// SIMATIC STEP 7 (V5.x) project Паллетайзер №2
// CPU: CPU 312
// station: P_ADR_BUS
// station: Hardware
// station: SIMATIC 300 Station
// program: S7 Program(2)

SYMBOL_TABLE
"FC2"	FC 2	FC 2	// Ручное управление
"FC3"	FC 3	FC 3	// Автоматическое управление
"КН1"	I 0.0	BOOL	// Кнопка ПУСК ВПЕРЕД устройства поддержания прокладки
"КН2"	I 0.1	BOOL	// Кнопка ПУСК НАЗАД устройства поддержания прокладки
"КН3"	I 0.2	BOOL	// Кнопка ПУСК ВПЕРЕД передвижная рама
"КН4"	I 0.3	BOOL	// Кнопка ПУСК НАЗАД передвижная рама
"КН5"	I 0.4	BOOL	// Кнопка ПУСК ВВЕРХ блокировка банок
"КН6"	I 0.5	BOOL	// Кнопка ПУСК ВНИЗ блокировка банок
"КН7"	I 0.6	BOOL	// Кнопка ПУСК ВВЕРХ штабелирующий лифт
"КН8"	I 0.7	BOOL	// Кнопка ПУСК ВНИЗ штабелирующий лифт
"КН9"	I 1.0	BOOL	// Кнопка ПУСК ВПЕРЕД выталкиватель
"КН10"	I 1.1	BOOL	// Кнопка ПУСК НАЗАД выталкиватель
"КН11"	I 1.2	BOOL	// Кнопка ПУСК ВВЕРХ лифт для паллет
"КН12"	I 1.3	BOOL	// Кнопка ПУСК ВНИЗ лифт для паллет
"6КВ1"	I 1.4	BOOL	// Лифт для паллет ВЕРХНЕЕ положение
"6КВ2"	I 1.5	BOOL	// Лифт для паллет НИЖНЕЕ положение
"КН15"	I 1.6	BOOL	// Кнопка ПУСК конвейера
"КН16"	I 1.7	BOOL	// Кнопка СТОП конвейера
"ПН17"	I 4.0	BOOL	// Переключатель РУЧНОЕ-АВТОМАТ
"КН18"	I 4.1	BOOL	// Кнопка ПУСК в автоматическом режиме
"КН17"	I 4.2	BOOL	// Аварийный СТОП
"4КВ2"	I 4.3	BOOL	// Штабелирующий лифт НИЖНЕЕ положение
"КН19"	I 4.4	BOOL	// Аварийный СТОП
"5КВ1"	I 4.5	BOOL	// Выталкиватель ПЕРЕДНЕЕ положение
"5КВ2"	I 4.6	BOOL	// Выталкиватель ЗАДДНЕЕ положение
"КН18а"	I 4.7	BOOL	// Кнопка Пуск в автоматическом режиме
"1КВ1"	I 5.0	BOOL	// Устройство поддержание прокладки ПЕРЕДНЕЕ положение
"1КВ2"	I 5.1	BOOL	// Устройство поддержание прокладки ЗАДНЕЕ положение
"1КВ3"	I 5.2	BOOL	// Устройство поддержание прокладки ВЕРХНЕЕ положение
"2КВ1"	I 5.3	BOOL	// Передвижная рама ПЕРЕДНЕЕ положение
"2КВ2"	I 5.4	BOOL	// Передвижная рама ЗАДДНЕЕ положение
"3КВ1"	I 5.5	BOOL	// Блокировка банок ВЕРХНЕЕ положение
"3КВ2"	I 5.6	BOOL	// Блокировка банок НИЖНЕЕ положение
"4КВ1"	I 5.7	BOOL	// Штабелирующий лифт ВЕРХНЕЕ положение
"8В1"	I 8.0	BOOL	// Наличие банки на накопительной ленте НАЧАЛО
"8В2"	I 8.1	BOOL	// Наличие банки на накопительной ленте СЕРЕДИНА
"8В3"	I 8.2	BOOL	// Наличие банки на накопительной ленте КОНЕЦ
"4КВ3"	I 8.3	BOOL	// Концевик счета слоев
"M0.0"	M 0.0	BOOL	// Меркер СТОП
"M0.1"	M 0.1	BOOL	// Меркер сброса таймера Т5
"M0.2"	M 0.2	BOOL	// Меркер счета слоев
"M2"	Q 12.0	BOOL	// Включение транспортера №2
"1КЛ1"	Q 12.2	BOOL	// Устройство поддержание прокладки ВПЕРЕД
"1КЛ2"	Q 12.3	BOOL	// Устройство поддержание прокладки НАЗАД
"2КЛ1"	Q 12.4	BOOL	// Передвижная рама ВПЕРЕД
"2КЛ2"	Q 12.5	BOOL	// Передвижная рама НАЗАД
"3КЛ1"	Q 12.6	BOOL	// Блокировка банок ВВЕРХ
"3КЛ2"	Q 12.7	BOOL	// Блокировка банок ВНИЗ
"4КЛ1"	Q 16.0	BOOL	// Штабелирующий лифт ВВЕРХ
"4КЛ2"	Q 16.1	BOOL	// Штабелирующий лифт ВНИЗ
"5КЛ1"	Q 16.2	BOOL	// Выталкиватель ВПЕРЕД
"5КЛ2"	Q 16.3	BOOL	// Выталкиватель НАЗАД
"6КЛ1"	Q 16.4	BOOL	// Лифт для паллет ВВЕРХ
"6КЛ2"	Q 16.5	BOOL	// Лифт для паллет ВНИЗ
"M1"	Q 16.6	BOOL	// Включение транспортера №1
"Zak"	Q 16.7	BOOL	// Блокировка включения закатки
"T1"	T 1	TIMER	// Задержка включения датчика 8В3
"T2"	T 2	TIMER	// Задержка включения датчика 8В2
"T3"	T 3	TIMER	// Включение движения выталкивателя НАЗАД
"T4"	T 4	TIMER	// Время перемещения штабелирующего лифта по времени
"T5"	T 5	TIMER	// Задержка перемещения блокировки банок ВВЕРХ
"T6"	T 6	TIMER
END_SYMBOL_TABLE

FUNCTION "FC2" : VOID	// FC 2
//Ручное управление
VERSION : 0.1
BEGIN
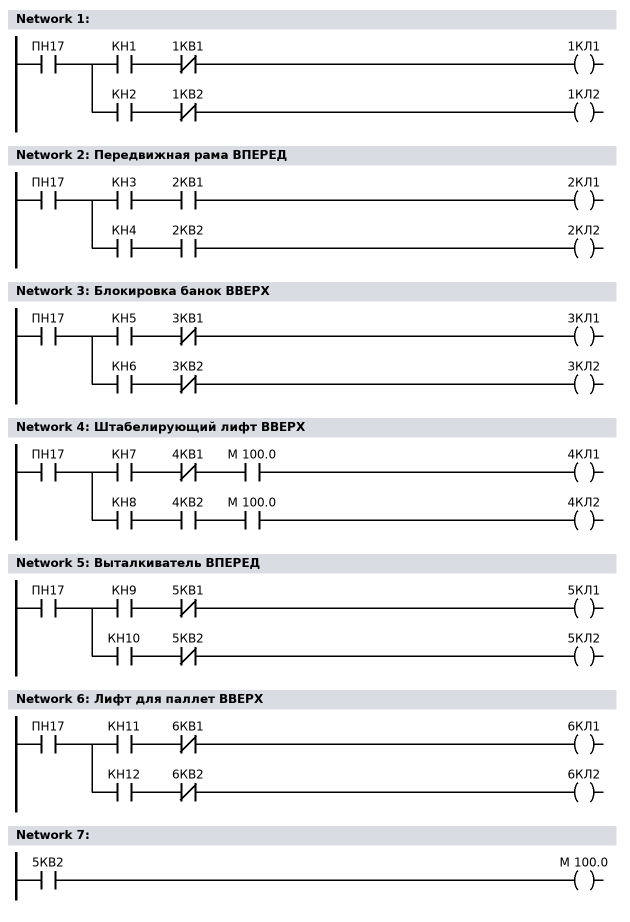
NETWORK
TITLE =
//Устройство поддержания прокладки
      A     "ПН17";
      =     L 0.0;
      A     L 0.0;
      A     "КН1";
      AN    "1КВ1";
      =     "1КЛ1";
      A     L 0.0;
      A     "КН2";
      AN    "1КВ2";
      =     "1КЛ2";
NETWORK
TITLE = Передвижная рама ВПЕРЕД
//Передвижная рама.
      A     "ПН17";
      =     L 0.0;
      A     L 0.0;
      A     "КН3";
      A     "2КВ1";
      =     "2КЛ1";
      A     L 0.0;
      A     "КН4";
      A     "2КВ2";
      =     "2КЛ2";
NETWORK
TITLE = Блокировка банок ВВЕРХ
//Устройство блокировки банок.
      A     "ПН17";
      =     L 0.0;
      A     L 0.0;
      A     "КН5";
      AN    "3КВ1";
      =     "3КЛ1";
      A     L 0.0;
      A     "КН6";
      AN    "3КВ2";
      =     "3КЛ2";
NETWORK
TITLE = Штабелирующий лифт ВВЕРХ
//Штабелирующий лифт.
      A     "ПН17";
      =     L 0.0;
      A     L 0.0;
      A     "КН7";
      AN    "4КВ1";
      A     M 100.0;
      =     "4КЛ1";
      A     L 0.0;
      A     "КН8";
      A     "4КВ2";
      A     M 100.0;
      =     "4КЛ2";
NETWORK
TITLE = Выталкиватель ВПЕРЕД
//Выталкиватель поддонов.
      A     "ПН17";
      =     L 0.0;
      A     L 0.0;
      A     "КН9";
      AN    "5КВ1";
      =     "5КЛ1";
      A     L 0.0;
      A     "КН10";
      AN    "5КВ2";
      =     "5КЛ2";
NETWORK
TITLE = Лифт для паллет ВВЕРХ
//Лифт для поддонов.
      A     "ПН17";
      =     L 0.0;
      A     L 0.0;
      A     "КН11";
      AN    "6КВ1";
      =     "6КЛ1";
      A     L 0.0;
      A     "КН12";
      AN    "6КВ2";
      =     "6КЛ2";
NETWORK
TITLE =
//Контроль заднего положения выталкивателя.
      A     "5КВ2";
      =     M 100.0;
END_FUNCTION

FUNCTION "FC3" : VOID	// FC 3
//Автоматическое управление
VERSION : 0.1
BEGIN
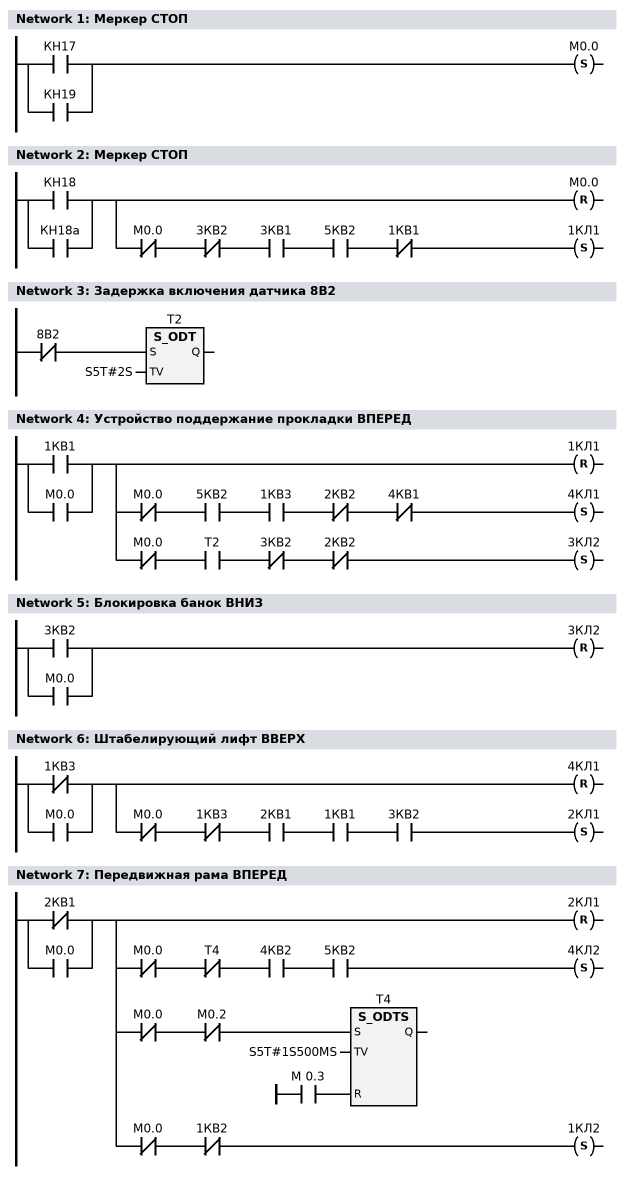
NETWORK
TITLE = Меркер СТОП
//Аварийный останов автоматического режима
      O     "КН17";
      O     "КН19";
      S     "M0.0";
NETWORK
TITLE = Меркер СТОП
//Запуск автоматического режима.
//Перемещение устройства поддержания прокладки ВПЕРЕД.
      O     "КН18";
      O     "КН18а";
      =     L 0.0;
      A     L 0.0;
      BLD   102;
      R     "M0.0";
      A     L 0.0;
      AN    "M0.0";
      AN    "3КВ2";
      A     "3КВ1";
      A     "5КВ2";
      AN    "1КВ1";
      S     "1КЛ1";
NETWORK
TITLE = Задержка включения датчика 8В2
      AN    "8В2";
      L     S5T#2S;
      SD    "T2";
      NOP   0;
      NOP   0;
      NOP   0;
      NOP   0;
NETWORK
TITLE = Устройство поддержание прокладки ВПЕРЕД
      O     "1КВ1";
      O     "M0.0";
      =     L 0.0;
      A     L 0.0;
      BLD   102;
      R     "1КЛ1";
      A     L 0.0;
      AN    "M0.0";
      A     "5КВ2";
      A     "1КВ3";
      AN    "2КВ2";
      AN    "4КВ1";
      S     "4КЛ1";
      A     L 0.0;
      AN    "M0.0";
      A     "T2";
      AN    "3КВ2";
      AN    "2КВ2";
      S     "3КЛ2";
NETWORK
TITLE = Блокировка банок ВНИЗ
      O     "3КВ2";
      O     "M0.0";
      R     "3КЛ2";
NETWORK
TITLE = Штабелирующий лифт ВВЕРХ
      ON    "1КВ3";
      O     "M0.0";
      =     L 0.0;
      A     L 0.0;
      BLD   102;
      R     "4КЛ1";
      A     L 0.0;
      AN    "M0.0";
      AN    "1КВ3";
      A     "2КВ1";
      A     "1КВ1";
      A     "3КВ2";
      S     "2КЛ1";
NETWORK
TITLE = Передвижная рама ВПЕРЕД
      ON    "2КВ1";
      O     "M0.0";
      =     L 0.0;
      A     L 0.0;
      BLD   102;
      R     "2КЛ1";
      A     L 0.0;
      AN    "M0.0";
      AN    "T4";
      A     "4КВ2";
      A     "5КВ2";
      S     "4КЛ2";
      A     L 0.0;
      AN    "M0.0";
      AN    "M0.2";
      L     S5T#1S500MS;
      SS    "T4";
      A     M 0.3;
      R     "T4";
      NOP   0;
      NOP   0;
      NOP   0;
      A     L 0.0;
      AN    "M0.0";
      AN    "1КВ2";
      S     "1КЛ2";
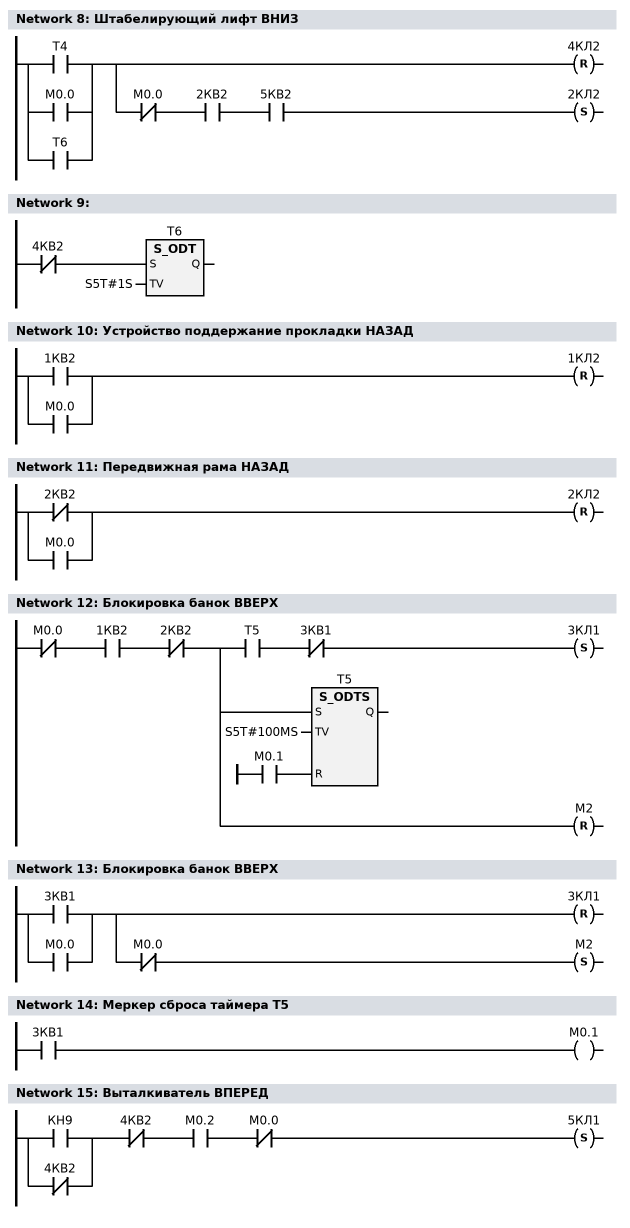
NETWORK
TITLE = Штабелирующий лифт ВНИЗ
      O     "T4";
      O     "M0.0";
      O     "T6";
      =     L 0.0;
      A     L 0.0;
      BLD   102;
      R     "4КЛ2";
      A     L 0.0;
      AN    "M0.0";
      A     "2КВ2";
      A     "5КВ2";
      S     "2КЛ2";
NETWORK
TITLE =
      AN    "4КВ2";
      L     S5T#1S;
      SD    "T6";
      NOP   0;
      NOP   0;
      NOP   0;
      NOP   0;
NETWORK
TITLE = Устройство поддержание прокладки НАЗАД
      O     "1КВ2";
      O     "M0.0";
      R     "1КЛ2";
NETWORK
TITLE = Передвижная рама НАЗАД
      ON    "2КВ2";
      O     "M0.0";
      R     "2КЛ2";
NETWORK
TITLE = Блокировка банок ВВЕРХ
      AN    "M0.0";
      A     "1КВ2";
      AN    "2КВ2";
      =     L 0.0;
      A     L 0.0;
      A     "T5";
      AN    "3КВ1";
      S     "3КЛ1";
      A     L 0.0;
      L     S5T#100MS;
      SS    "T5";
      A     "M0.1";
      R     "T5";
      NOP   0;
      NOP   0;
      NOP   0;
      A     L 0.0;
      BLD   102;
      R     "M2";
NETWORK
TITLE = Блокировка банок ВВЕРХ
      O     "3КВ1";
      O     "M0.0";
      =     L 0.0;
      A     L 0.0;
      BLD   102;
      R     "3КЛ1";
      A     L 0.0;
      AN    "M0.0";
      S     "M2";
NETWORK
TITLE = Меркер сброса таймера Т5
      A     "3КВ1";
      =     "M0.1";
NETWORK
TITLE = Выталкиватель ВПЕРЕД
      A(;
      O     "КН9";
      ON    "4КВ2";
      );
      AN    "4КВ2";
      A     "M0.2";
      AN    "M0.0";
      S     "5КЛ1";
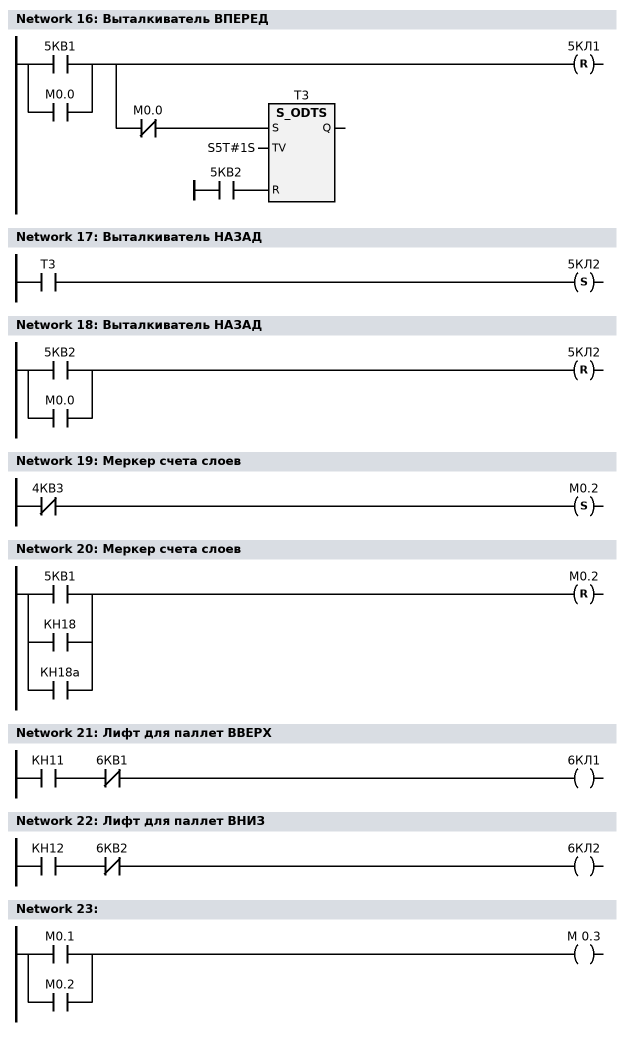
NETWORK
TITLE = Выталкиватель ВПЕРЕД
      O     "5КВ1";
      O     "M0.0";
      =     L 0.0;
      A     L 0.0;
      BLD   102;
      R     "5КЛ1";
      A     L 0.0;
      AN    "M0.0";
      L     S5T#1S;
      SS    "T3";
      A     "5КВ2";
      R     "T3";
      NOP   0;
      NOP   0;
      NOP   0;
NETWORK
TITLE = Выталкиватель НАЗАД
      A     "T3";
      S     "5КЛ2";
NETWORK
TITLE = Выталкиватель НАЗАД
      O     "5КВ2";
      O     "M0.0";
      R     "5КЛ2";
NETWORK
TITLE = Меркер счета слоев
      AN    "4КВ3";
      S     "M0.2";
NETWORK
TITLE = Меркер счета слоев
      O     "5КВ1";
      O     "КН18";
      O     "КН18а";
      R     "M0.2";
NETWORK
TITLE = Лифт для паллет ВВЕРХ
      A     "КН11";
      AN    "6КВ1";
      =     "6КЛ1";
NETWORK
TITLE = Лифт для паллет ВНИЗ
      A     "КН12";
      AN    "6КВ2";
      =     "6КЛ2";
NETWORK
TITLE =
      O     "M0.1";
      O     "M0.2";
      =     M 0.3;
END_FUNCTION

ORGANIZATION_BLOCK OB 1
TITLE = "Main Program Sweep (Cycle)"
VERSION : 0.1
VAR_TEMP
  OB1_EV_CLASS : BYTE ;	//Bits 0-3 = 1 (Coming event), Bits 4-7 = 1 (Event class 1)
  OB1_SCAN_1 : BYTE ;	//1 (Cold restart scan 1 of OB 1), 3 (Scan 2-n of OB 1)
  OB1_PRIORITY : BYTE ;	//Priority of OB Execution
  OB1_OB_NUMBR : BYTE ;	//1 (Organization block 1, OB1)
  OB1_RESERVED_1 : BYTE ;	//Reserved for system
  OB1_RESERVED_2 : BYTE ;	//Reserved for system
  OB1_PREV_CYCLE : INT ;	//Cycle time of previous OB1 scan (milliseconds)
  OB1_MIN_CYCLE : INT ;	//Minimum cycle time of OB1 (milliseconds)
  OB1_MAX_CYCLE : INT ;	//Maximum cycle time of OB1 (milliseconds)
  OB1_DATE_TIME : DATE_AND_TIME ;	//Date and time OB1 started
END_VAR
BEGIN
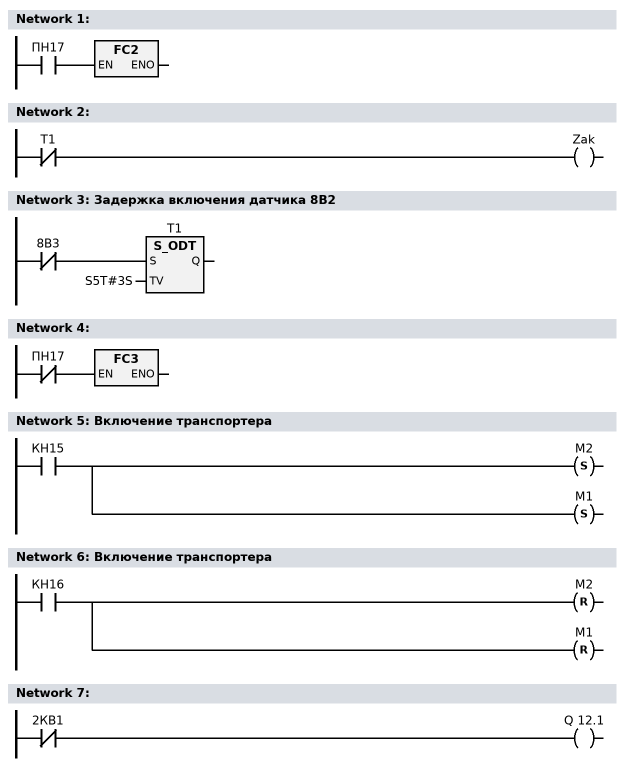
NETWORK
TITLE =
//Включение режима ручного управления.
      A     "ПН17";
      JNB   _001;
      CALL  "FC2";
_001: NOP   0;
NETWORK
TITLE =
      AN    "T1";
      =     "Zak";
NETWORK
TITLE = Задержка включения датчика 8В2
      AN    "8В3";
      L     S5T#3S;
      SD    "T1";
      NOP   0;
      NOP   0;
      NOP   0;
      NOP   0;
NETWORK
TITLE =
//Включение режима автоматического управления.
      AN    "ПН17";
      JNB   _002;
      CALL  "FC3";
_002: NOP   0;
NETWORK
TITLE = Включение транспортера
//Включение транспортеров.
      A     "КН15";
      S     "M2";
      S     "M1";
NETWORK
TITLE = Включение транспортера
//Выключение транспортеров.
      A     "КН16";
      R     "M2";
      R     "M1";
NETWORK
TITLE =
      AN    "2КВ1";
      =     Q 12.1;
END_ORGANIZATION_BLOCK
